(* IEC 61131-3 sources: lc3-wifi-kurs/src/example_1_i2c_digital, 1 file *)

(* ---- i2c_digital.iecst ---- *)
PROGRAM Program_I2C_Digital
	VAR
		i2c_handle : DINT := -1;
		pinValues_1 : ARRAY [0..7] OF BOOL;
	END_VAR

	IF i2c_handle < 0 THEN
		i2c_handle := I2C_open(bus_id := 1);
	ELSE
		pinValues_1 := I2C_PCF8574_read(fd := i2c_handle, address := I2C_ADDRESSES#PCF8574_INPUT_1);
		I2C_PCF8574_write(fd := i2c_handle, address := I2C_ADDRESSES#PCF8574_OUTPUT_1, pin_values := pinValues_1);
	END_IF;
END_PROGRAM
